{attribute addProperty BoxType "EJ5101-0000-0016"}
{attribute addProperty Id "ControlAT %Q*Control_38B054C81621Set_counter_valueAT %Q*UINT16217"}
{attribute addProperty CRC "57679667"}
{attribute addProperty SizeInBites "32"}
{attribute addProperty SizeInBytes "4"}
TYPE ENC_Control_compact_03701F33 :
STRUCT
	{attribute addProperty Name "Control"}
	Control AT %Q* : Control_38B054C8;
	{attribute addProperty Name "Set_counter_value"}
	Set_counter_value AT %Q* : UINT;
END_STRUCT
END_TYPE

(* stored: Version 1.2.0.0, ProductVersion 3.1.4024.9
   DUT ENC_Control_compact_03701F33: Id {4020f17d-866d-4298-a2ea-be3b640de747} *)
